FUNCTION_BLOCK MCCPower_HMI (* Service Interface Function Block Type *)
  (* Standard: 61499-2 *)
  (* Version 0.0, 3/8/2024, SESA371406, Schneider Electric, template *)
  PACKAGE SE.Nereda;
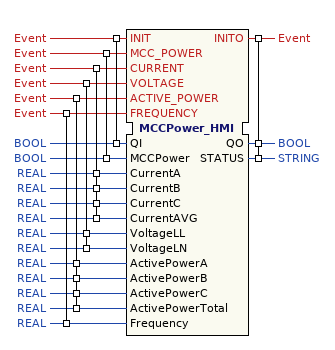
  EVENT_INPUT
    INIT WITH QI;
    MCC_POWER WITH MCCPower;
    CURRENT WITH CurrentA, CurrentB, CurrentC, CurrentAVG;
    VOLTAGE WITH VoltageLL, VoltageLN;
    ACTIVE_POWER WITH ActivePowerA, ActivePowerB, ActivePowerC, ActivePowerTotal;
    FREQUENCY WITH Frequency;
  END_EVENT
  EVENT_OUTPUT
    INITO WITH QO, STATUS;
  END_EVENT
  VAR_INPUT
    QI : BOOL;
    MCCPower : BOOL;
    CurrentA : REAL;
    CurrentB : REAL;
    CurrentC : REAL;
    CurrentAVG : REAL;
    VoltageLL : REAL;
    VoltageLN : REAL;
    ActivePowerA : REAL;
    ActivePowerB : REAL;
    ActivePowerC : REAL;
    ActivePowerTotal : REAL;
    Frequency : REAL;
  END_VAR
  VAR_OUTPUT
    QO : BOOL; (* Event Output Qualifier *)
    STATUS : STRING; (* Service Status *)
  END_VAR
  SERVICE /
    SEQUENCE 
    END_SEQUENCE
  END_SERVICE
END_FUNCTION_BLOCK
